PROGRAM ModbusTcp
Var
    MW  : FB_SplitRealToWords_IEEE754;
    MW1  : FB_SplitUlintToWords;
(*
   mySimpleTcpServer: FbMbSimpleServerTcp :=(  xOpen           := TRUE,  wPort := 2000,bUnitId := 1,
                                              utKeepAlive     := (xEnable      := TRUE, //  Switch keep-alive mechanism on
                                                                       tMaxIdleTime := T#5S, //  Maximum time of inactivity
                                                                        tInterval    := T#2S, //  Interval between two successive KA-Packets
                                                                     udiProbes    := 5 ));    //  Number of KA retry before giving up
*)
END_VAR


(* 
//--- Call the server --------------------------------------------- 
mySimpleTcpServer(  awHoldingRegisters  := GVL_DataBaseStructures.AX_StructModbusTCP    ); 
 *)

END_PROGRAM

(* stored: Version 1.1.0.1, ProductVersion 3.1.4024.11
   POU ModbusTcp: Id {fa9b2688-9ad5-4e00-88e3-495a92adddcc}, SpecialFunc None *)
